{attribute 'qualified_only'}
{attribute 'to_string'}
TYPE E_TakeOverState:
(**************************************************************************************
 * 	Application		:	BoxControl Framework
 *	Revision		:	$Revision: 404529 $
 *	Revision date	:	$Date: 2018-04-23 08:21:38 +0200 (Mo., 23 Apr 2018) $
 *	Last changed by	:	$Author: b7bolm $
 *	URL				:	$URL: http://almscdc.swisslog.com/repo/SWPD/Development/BoxControlFramework/20_Release/trunk/01_Software/BCF/BCF/JumpStart/20_Product/10_App/12_E_Functions/10_Lib/10_Conv/10_Functions/01_DUTs/E_TakeOverState.TcDUT $
 *
 *	Purpose			:	TakeOver states
 *
 * ------------------------------------------------------------------------------------
 *	Copyright Swisslog [IP AG], Switzerland. All rights reserved.
 * 
 * ------------------------------------------------------------------------------------
 *	
 * 	Revision History: 
 *
 * 	VERSION			DATE			INITIALS			DESCRIPTION
 *	0.1				01.01.2001		swl					Example 
 *
 **************************************************************************************)
(
	UNDEFINED			:= 0,
	IDLE				:= 1,
	READY				:= 2,
	ACTIVE				:= 4,
	STOP				:= 5,
	INTERRUPTED			:= 6,
	COMPLETE			:= 7
);
END_TYPE

(* stored: Version 1.1.0.1, ProductVersion 3.1.4024.9
   DUT E_TakeOverState: Id {cffbc3d4-cc12-4cea-a67c-0e64200d2d18} *)
